SUBAPPLICATION Uebung_053 (* DigitalInput_I1-_I4 auf DigitalOutput_Q1-_Q4 *)
  (* Standard: 61499-2 *)
  (* Version 1.0, 2023-10-23, franz *)
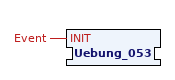
  EVENT_INPUT
    INIT;
  END_EVENT
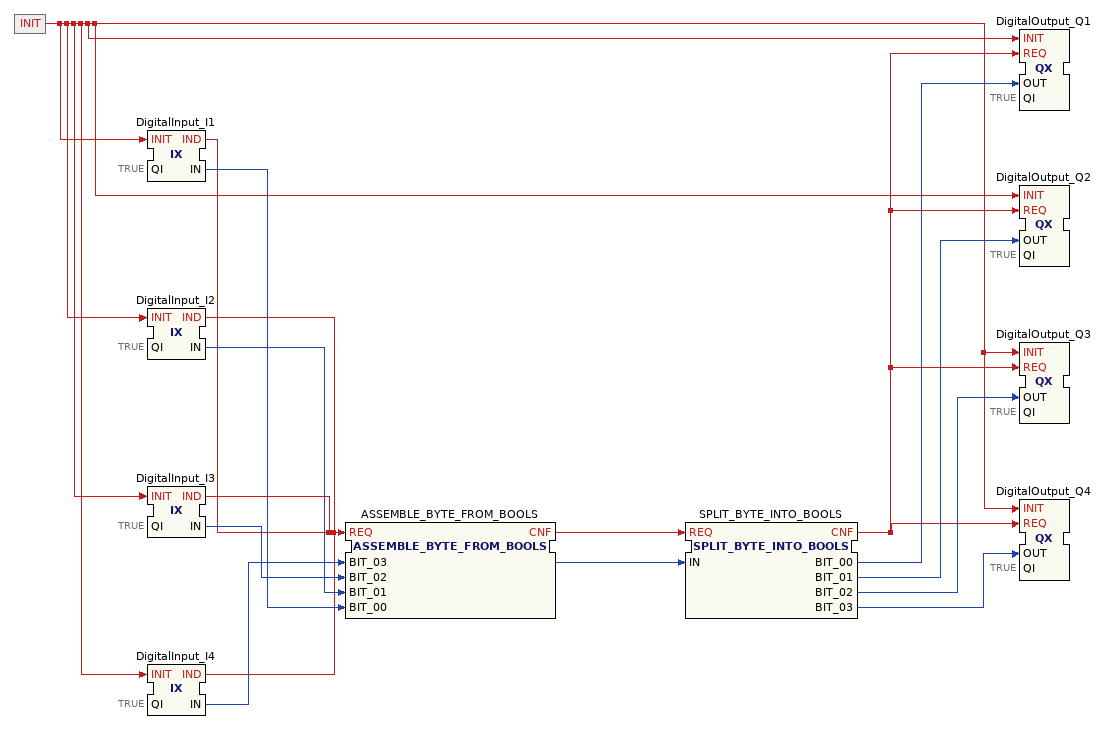
  FBS
    DigitalOutput_Q1 : QX(QI := TRUE);
    DigitalInput_I1 : IX(QI := TRUE);
    DigitalOutput_Q2 : QX(QI := TRUE);
    DigitalInput_I2 : IX(QI := TRUE);
    DigitalOutput_Q3 : QX(QI := TRUE);
    DigitalInput_I3 : IX(QI := TRUE);
    DigitalOutput_Q4 : QX(QI := TRUE);
    DigitalInput_I4 : IX(QI := TRUE);
    ASSEMBLE_BYTE_FROM_BOOLS : ASSEMBLE_BYTE_FROM_BOOLS;
    SPLIT_BYTE_INTO_BOOLS : SPLIT_BYTE_INTO_BOOLS;
  END_FBS
  EVENT_CONNECTIONS
    INIT TO DigitalInput_I1.INIT;
    INIT TO DigitalInput_I2.INIT;
    INIT TO DigitalInput_I3.INIT;
    INIT TO DigitalInput_I4.INIT;
    INIT TO DigitalOutput_Q1.INIT;
    INIT TO DigitalOutput_Q2.INIT;
    INIT TO DigitalOutput_Q3.INIT;
    INIT TO DigitalOutput_Q4.INIT;
    ASSEMBLE_BYTE_FROM_BOOLS.CNF TO SPLIT_BYTE_INTO_BOOLS.REQ;
    DigitalInput_I1.IND TO ASSEMBLE_BYTE_FROM_BOOLS.REQ;
    DigitalInput_I2.IND TO ASSEMBLE_BYTE_FROM_BOOLS.REQ;
    DigitalInput_I3.IND TO ASSEMBLE_BYTE_FROM_BOOLS.REQ;
    DigitalInput_I4.IND TO ASSEMBLE_BYTE_FROM_BOOLS.REQ;
    SPLIT_BYTE_INTO_BOOLS.CNF TO DigitalOutput_Q1.REQ;
    SPLIT_BYTE_INTO_BOOLS.CNF TO DigitalOutput_Q2.REQ;
    SPLIT_BYTE_INTO_BOOLS.CNF TO DigitalOutput_Q3.REQ;
    SPLIT_BYTE_INTO_BOOLS.CNF TO DigitalOutput_Q4.REQ;
  END_CONNECTIONS
  DATA_CONNECTIONS
    ASSEMBLE_BYTE_FROM_BOOLS. TO SPLIT_BYTE_INTO_BOOLS.IN;
    SPLIT_BYTE_INTO_BOOLS.BIT_00 TO DigitalOutput_Q1.OUT;
    SPLIT_BYTE_INTO_BOOLS.BIT_01 TO DigitalOutput_Q2.OUT;
    SPLIT_BYTE_INTO_BOOLS.BIT_02 TO DigitalOutput_Q3.OUT;
    SPLIT_BYTE_INTO_BOOLS.BIT_03 TO DigitalOutput_Q4.OUT;
    DigitalInput_I4.IN TO ASSEMBLE_BYTE_FROM_BOOLS.BIT_03;
    DigitalInput_I3.IN TO ASSEMBLE_BYTE_FROM_BOOLS.BIT_02;
    DigitalInput_I2.IN TO ASSEMBLE_BYTE_FROM_BOOLS.BIT_01;
    DigitalInput_I1.IN TO ASSEMBLE_BYTE_FROM_BOOLS.BIT_00;
  END_CONNECTIONS
END_SUBAPPLICATION
